// TIA Portal V17 export
// export: Created 2021-12-03T08:13:06.0675145Z, ExportSetting WithDefaults, DisplayName Totally Integrated Automation Portal, DisplayVersion V17, DisplayName TIA Portal Openness, DisplayVersion V17, DisplayName TIA Portal Version Control Interface, DisplayVersion V17, DisplayName STEP 7 Professional, DisplayVersion V17, DisplayName STEP 7 Safety, DisplayVersion V17, DisplayName WinCC Advanced, DisplayVersion V17
DATA_BLOCK "GDB_ConvCtrl"   // DB500
VERSION : 0.1
// stored: AutoNumber false, IsOnlyStoredInLoadMemory false, IsWriteProtectedInAS false
   VAR
      FrqConv : Struct
         reqForward : Bool;   // Прямое направление
         reqBackward : Bool;   // Обратное направление
         reqSpeed : Int;   // Запрашиваемая скорость
         reqRampe : Int;   // Запрашиваемая рампа
         Fault : Bool;   // Ошибка
         FaultNumber : Int;   // Номер ошибки
         ActSpeed : Int;   // Текущая скорость
         ActCurrent : Int;   // Текущий ток
      END_STRUCT;
      LowSpeed : Bool;
      FrqConvPwrOn : Bool;
      SpeedCalculation : Struct
         SpeedMov : Int;
         TimeMov : Int;
         DistanceX10 : Int;
         SelDistance : Int;
      END_STRUCT;
      SR : Struct
         FrqConvPwrOn : Bool;
      END_STRUCT;
      Trig : Struct
         P_SlowFwd : Bool;
         P_SlowBwd : Bool;
         N_SlowFwd : Bool;
         N_SlowBwd : Bool;
         P_StrtFwd : Bool;
         P_StrtBwd : Bool;
      END_STRUCT;
      Animation : Struct
         Speed : Int;
         CalcBit : Bool;
         N_Trig : Bool;
         SR : Bool;
         Value : Real;
      END_STRUCT;
   END_VAR
BEGIN
END_DATA_BLOCK
